// TwinCAT 3 PLC project Altator_Program
// ProgramVersion: 3.1.4026.17
// CompilerDefines: VISU_USEPROPERTYINFO
// libraries:
//   Tc2_Math, * (Beckhoff Automation GmbH)
//   Tc2_Standard, * (Beckhoff Automation GmbH)
//   Tc2_System, * (Beckhoff Automation GmbH)
// project tree:
//   / GlobalTextList.TcGTLO, PlcTask.TcTTO, TrendRefreshTask.TcTTO, Visualization Manager.TcVMO (not stored), VISU_TASK.TcTTO
//   GVLs/ GVL_Data.TcGVL
//   POUs/ FB_Gauge.TcPOU, MAIN.TcPOU, POU_TrendLine.TcPOU
//   VISUs/ Visualization.TcVIS
// real-time tasks:
//   TASK PlcTask: cycle T#10ms, priority 20, ADS port 350
//   TASK VISU_TASK: cycle T#200000us, priority 30, ADS port 351
//   TASK TrendRefreshTask: cycle T#120ms, priority 31, ADS port 352
// I/O:
//   DEVICE Device 1 (EtherCAT), AmsNetId 10.0.0.23.2.1
//     Term 1 (EK1200) [EK1200-5000 EtherCAT Power supply (2A E-Bus)]
//       Term 2 (EL1014) [EL1014 4Ch. Dig. Input 24V, 10µs]
//       Term 3 (EL2004) [EL2004 4Ch. Dig. Output 24V, 0.5A]
//       Term 4 (EL3022) [EL3022 2Ch. Ana. Input 4-20mA DIFF]
//       Term 5 (EL4008) [EL4008 8Ch. Ana. Output 0-10V, 12bit]
//       Term 6 (EL3314-0010) [EL3314-0010 4Ch. Ana Input Thermocouple (TC), High Precision]
//       Term 7 (EL1918) [EL1918, 8Ch. Safety Input 24V, TwinSAFE]
//         modules: Module 1 (FSOE), Module 2 (FSLOGIC)
//       Term 8 (EL2904) [EL2904, 4 Ch. Safety Output 24V, 0.5A, TwinSAFE]
//         modules: Module 1 (FSOES), Module 2 (DO)
//       Term 9 (EL9011) [EL9011 End Terminal]
// variable links:
//   Altator_Program/Altator_Program Instance <-> Device 1 (EtherCAT)/Term 1 (EK1200)/Term 4 (EL3022)
//     PlcTask Inputs/MAIN.fb_Gauge_01.nRawVoltage <-> AI Standard Channel 1/Value

CONFIGURATION Altator_Program
    RESOURCE PLC ON TwinCAT3
        TASK PlcTask(INTERVAL := T#10ms, PRIORITY := 20);
        TASK TrendRefreshTask(INTERVAL := T#120ms, PRIORITY := 31);
        TASK VISU_TASK(INTERVAL := T#200000us, PRIORITY := 30);
        PROGRAM MAIN WITH PlcTask : MAIN;
        PROGRAM VisuElems_Visu_Prg WITH VISU_TASK : VisuElems.Visu_Prg;
    END_RESOURCE
END_CONFIGURATION

// ---- GVLs/GVL_Data.TcGVL
{attribute 'qualified_only'}
VAR_GLOBAL
	fAnalogData : REAL;
	fTestDelta : REAL;
	bTrendStatus : BOOL;
END_VAR

VAR_GLOBAL CONSTANT
	aiTrendArrayMax : INT;
END_VAR

// ---- POUs/MAIN.TcPOU
PROGRAM MAIN
VAR
	fb_Gauge_01 : FB_Gauge; // 01 moniker used in case future gauges are added
END_VAR

fb_Gauge_01();

END_PROGRAM

// ---- POUs/FB_Gauge.TcPOU
FUNCTION_BLOCK FB_Gauge
VAR_INPUT
	nRawVoltage AT %I* : INT; // Raw data input to EL3102
END_VAR
VAR_OUTPUT
	rPressureTorr : REAL; // Pressure value
END_VAR
VAR
	
	nScaledVoltage : REAL; // Scratch variable for converting voltage to real
	bStatus : BOOL ; 
END_VAR

nScaledVoltage := (TO_LREAL(nRawVoltage) / 32767.0) * 10.0;

IF (nScaledVoltage>= 0.375) AND (nScaledVoltage<= 2.842) THEN
rPressureTorr := -0.02585 
               + (0.03767 * nScaledVoltage) 
               + (0.04563 * EXPT(nScaledVoltage,2))
               + (0.1151  * EXPT(nScaledVoltage,3)) 
               + (-0.04158 * EXPT(nScaledVoltage,4)) 
               + (0.008737 * EXPT(nScaledVoltage,5));

ELSIF (nScaledVoltage> 2.842) AND (nScaledVoltage<= 4.945) THEN
	rPressureTorr := (0.1031+(nScaledVoltage*(-0.02322))
					+ (0.07227*EXPT(nScaledVoltage,2)))
					/ (1+(-0.3986*nScaledVoltage)
					+(0.07438*(EXPT(nScaledVoltage,2)))
					+(-0.006866*(EXPT(nScaledVoltage,3))));

ELSIF  (nScaledVoltage> 4.945) AND (nScaledVoltage<= 5.569) THEN
	rPressureTorr := 100.624 + (nScaledVoltage * (-20.5623));

ELSE
	bStatus := FALSE;
END_IF

END_FUNCTION_BLOCK

// ---- POUs/POU_TrendLine.TcPOU
FUNCTION_BLOCK POU_TrendLine
VAR
	aiLoopIndex : DINT;
	ArrayTrend : ARRAY[1..GVL_Data.aiTrendArrayMax]OF REAL;
	ArrayTrendDisp : ARRAY[1..GVL_Data.aiTrendArrayMax]OF REAL;
END_VAR

// Trend array loop
FOR aiLoopIndex := 1 TO (GVL_Data.aiTrendArrayMax-1) DO
	ArrayTrend[aiLoopIndex] := ArrayTrend[aiLoopIndex + 1];
	
END_FOR

ArrayTrend[GVL_Data.aiTrendArrayMax] := GVL_Data.fAnalogData;

// When Pause is OFF, Update the ArrayTrendDisp Array
IF NOT GVL_Data.bTrendStatus THEN
	FOR aiLoopIndex := 1 TO GVL_Data.aiTrendArrayMax DO
		ArrayTrendDisp[aiLoopIndex] := ArrayTrend[aiLoopIndex + 1];
	END_FOR
END_IF

END_FUNCTION_BLOCK

// ---- GlobalTextList.TcGTLO
TEXTLIST GlobalTextList
  892 = 'Pirani Gauge Pressure'
  206 = 'Start'
END_TEXTLIST

// ---- VISUs/Visualization.TcVIS
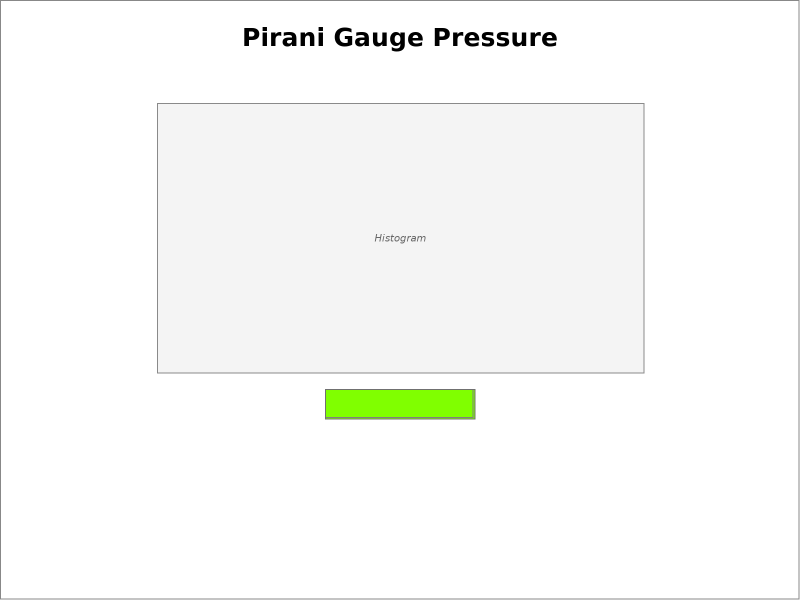
VISUALIZATION Visualization  // 800x600
    Label (160,5 480x64), "Pirani Gauge Pressure"
    Histogram (157,103 487x270), scale format: %.1f, scale 0..100
    Button (325,389 150x30)
END_VISUALIZATION
